// Return TRUE on a successful (Ok) result.
// Optionally carries the value over to nOut for further processing.
FUNCTION IsOk : BOOL
VAR_INPUT
    nIn : Result; // Result variable to check for success
END_VAR
VAR_OUTPUT
    nOut : Result; // Carries the input value for further use
END_VAR

IsOk := nIn > 0;
nOut := nIn;

END_FUNCTION

(* stored: Version 1.1.0.1
   POU IsOk: Id {a86826be-b52a-46f1-b35e-fa89d49ee7eb}, SpecialFunc None *)
